TYPE ST_DebugStation :
STRUCT
		stGblDBStnParam		: ST_DebugStationSeqParam;
		fbDBStnSeq			: FB_DebugStationSeq;
END_STRUCT
END_TYPE

(* stored: Version 1.1.0.1, ProductVersion 3.1.4022.18
   DUT ST_DebugStation: Id {7f94506e-a20d-4429-a361-d46a6509b87b} *)
